# EPICS autosave request: soft_iocs/flir_cameras/iocBoot/iocflir_c_mono1/auto_settings.req
file "spinnaker_settings.req",            P=$(P),  R=cam1:
file "NDStdArrays_settings.req",          P=$(P),  R=image1:
file "commonPlugin_settings.req",         P=$(P)
file "ffmpegServer_settings.req",         P=$(P),  R=ffmstream1:
